TYPE EventMessageHMI :
STRUCT
  timestamp: LString;
  path: LString;
  message: LString;
  level: EventLevel;
END_STRUCT
END_TYPE

(* stored: Version 1.1.0.1, ProductVersion 3.1.4024.9
   DUT EventMessageHMI: Id {c2876103-f28c-4070-9615-95f28d277a60} *)
